PROGRAM main
  VAR
    Emergency_PB AT %IX0.0 : BOOL;
    Start_PB AT %IX0.1 : BOOL;
    Stop_PB AT %IX0.2 : BOOL;
    Fill_PositionSensor AT %IX0.4 : BOOL;
    Fill_LevelSensor AT %IX0.5 : BOOL;
    Cap_PresentSensor AT %IX0.6 : BOOL;
    NA_LabelSensor AT %IX0.7 : BOOL;
    To_M_Conv_Sensor AT %IX1.0 : BOOL;
    CaseFull_Sensor AT %IX1.1 : BOOL;
    M0 AT %IX1.2 : BOOL;
    M1 AT %IX1.3 : BOOL;
    Safety_Trip AT %IX1.4 : BOOL;
    Fill_Active AT %IX1.5 : BOOL;
    Label_PositionSensor AT %IX1.6 : BOOL;
    Reset_PB AT %IX1.7 : BOOL;
    InfeedConv_M AT %QX0.0 : BOOL;
    MainConv_M AT %QX0.1 : BOOL;
    FillValve AT %QX0.2 : BOOL;
    CapHead_M AT %QX0.3 : BOOL;
    LabelApplicator_M AT %QX0.4 : BOOL;
    RejectAcctuator_1 AT %QX0.5 : BOOL;
    RejectAcctuator_2 AT %QX0.6 : BOOL;
    TransferAcctuator AT %QX0.7 : BOOL;
    CasePacker_M AT %QX1.0 : BOOL;
    StackLight_Green AT %QX1.1 : BOOL;
    StackLight_Red AT %QX1.2 : BOOL;
    StackLight_Yellow AT %QX1.3 : BOOL;
    Alarm_Buzzer AT %QX1.4 : BOOL;
    Siren AT %QX1.5 : BOOL;
    TP0 : TP;
    TP1 : TP;
    TP2 : TP;
    TP3 : TP;
    CTU0 : CTU;
    TON0 : TON;
    TON1 : TON;
    TON2 : TON;
    RS0 : RS;
    RS1 : RS;
    RS2 : RS;
  END_VAR

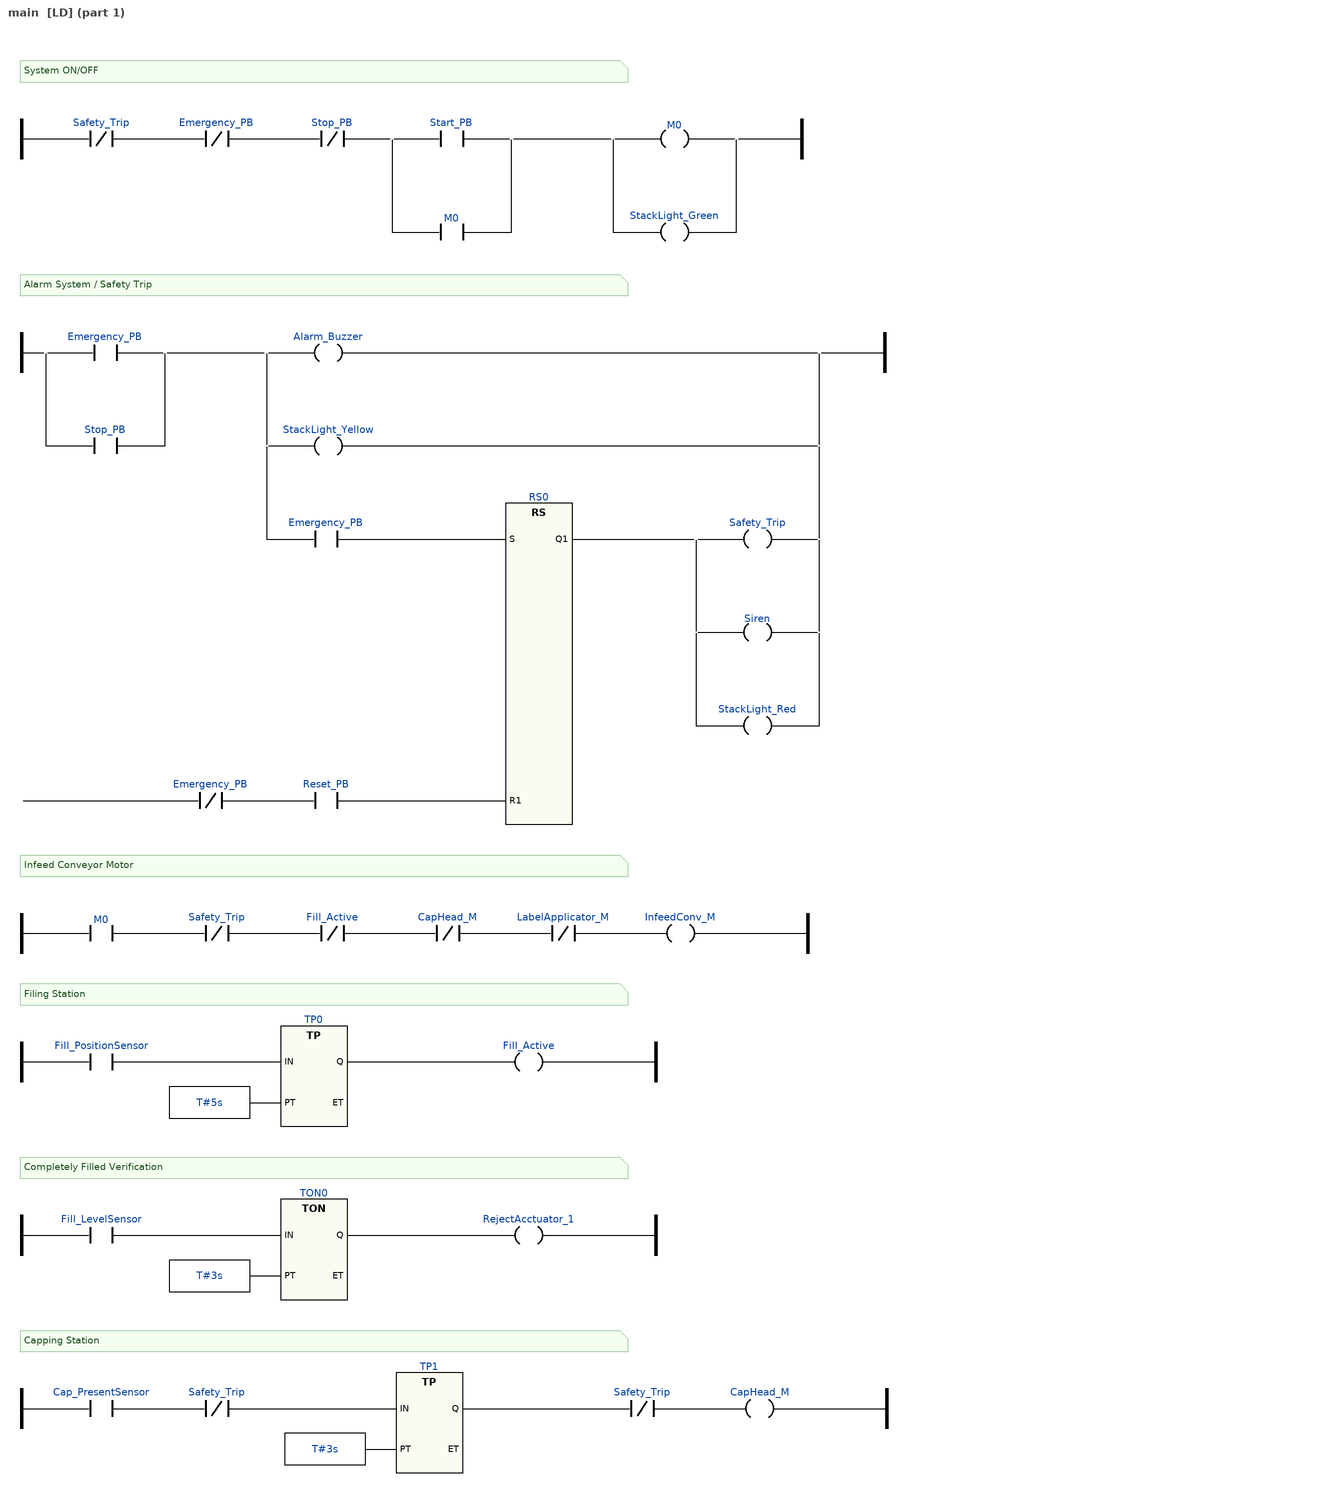
(* LD diagram, written out as Structured Text *)
(* System ON/OFF *)
M0 := NOT Safety_Trip AND NOT Emergency_PB AND NOT Stop_PB AND (Start_PB OR M0);
StackLight_Green := NOT Safety_Trip AND NOT Emergency_PB AND NOT Stop_PB AND (Start_PB OR M0);
(* Alarm System / Safety Trip *)
Alarm_Buzzer := Emergency_PB OR Stop_PB;
StackLight_Yellow := Emergency_PB OR Stop_PB;
RS0(S := (Emergency_PB OR Stop_PB) AND Emergency_PB, R1 := NOT Emergency_PB AND Reset_PB);
Safety_Trip := RS0.Q1;
Siren := RS0.Q1;
StackLight_Red := RS0.Q1;
(* Infeed Conveyor Motor *)
InfeedConv_M := M0 AND NOT Safety_Trip AND NOT Fill_Active AND NOT CapHead_M AND NOT LabelApplicator_M;
(* Filing Station *)
TP0(IN := Fill_PositionSensor, PT := T#5s);
Fill_Active := TP0.Q;
(* Completely Filled Verification *)
TON0(IN := Fill_LevelSensor, PT := T#3s);
RejectAcctuator_1 := TON0.Q;
(* Capping Station *)
TP1(IN := Cap_PresentSensor AND NOT Safety_Trip, PT := T#3s);
CapHead_M := TP1.Q AND NOT Safety_Trip;
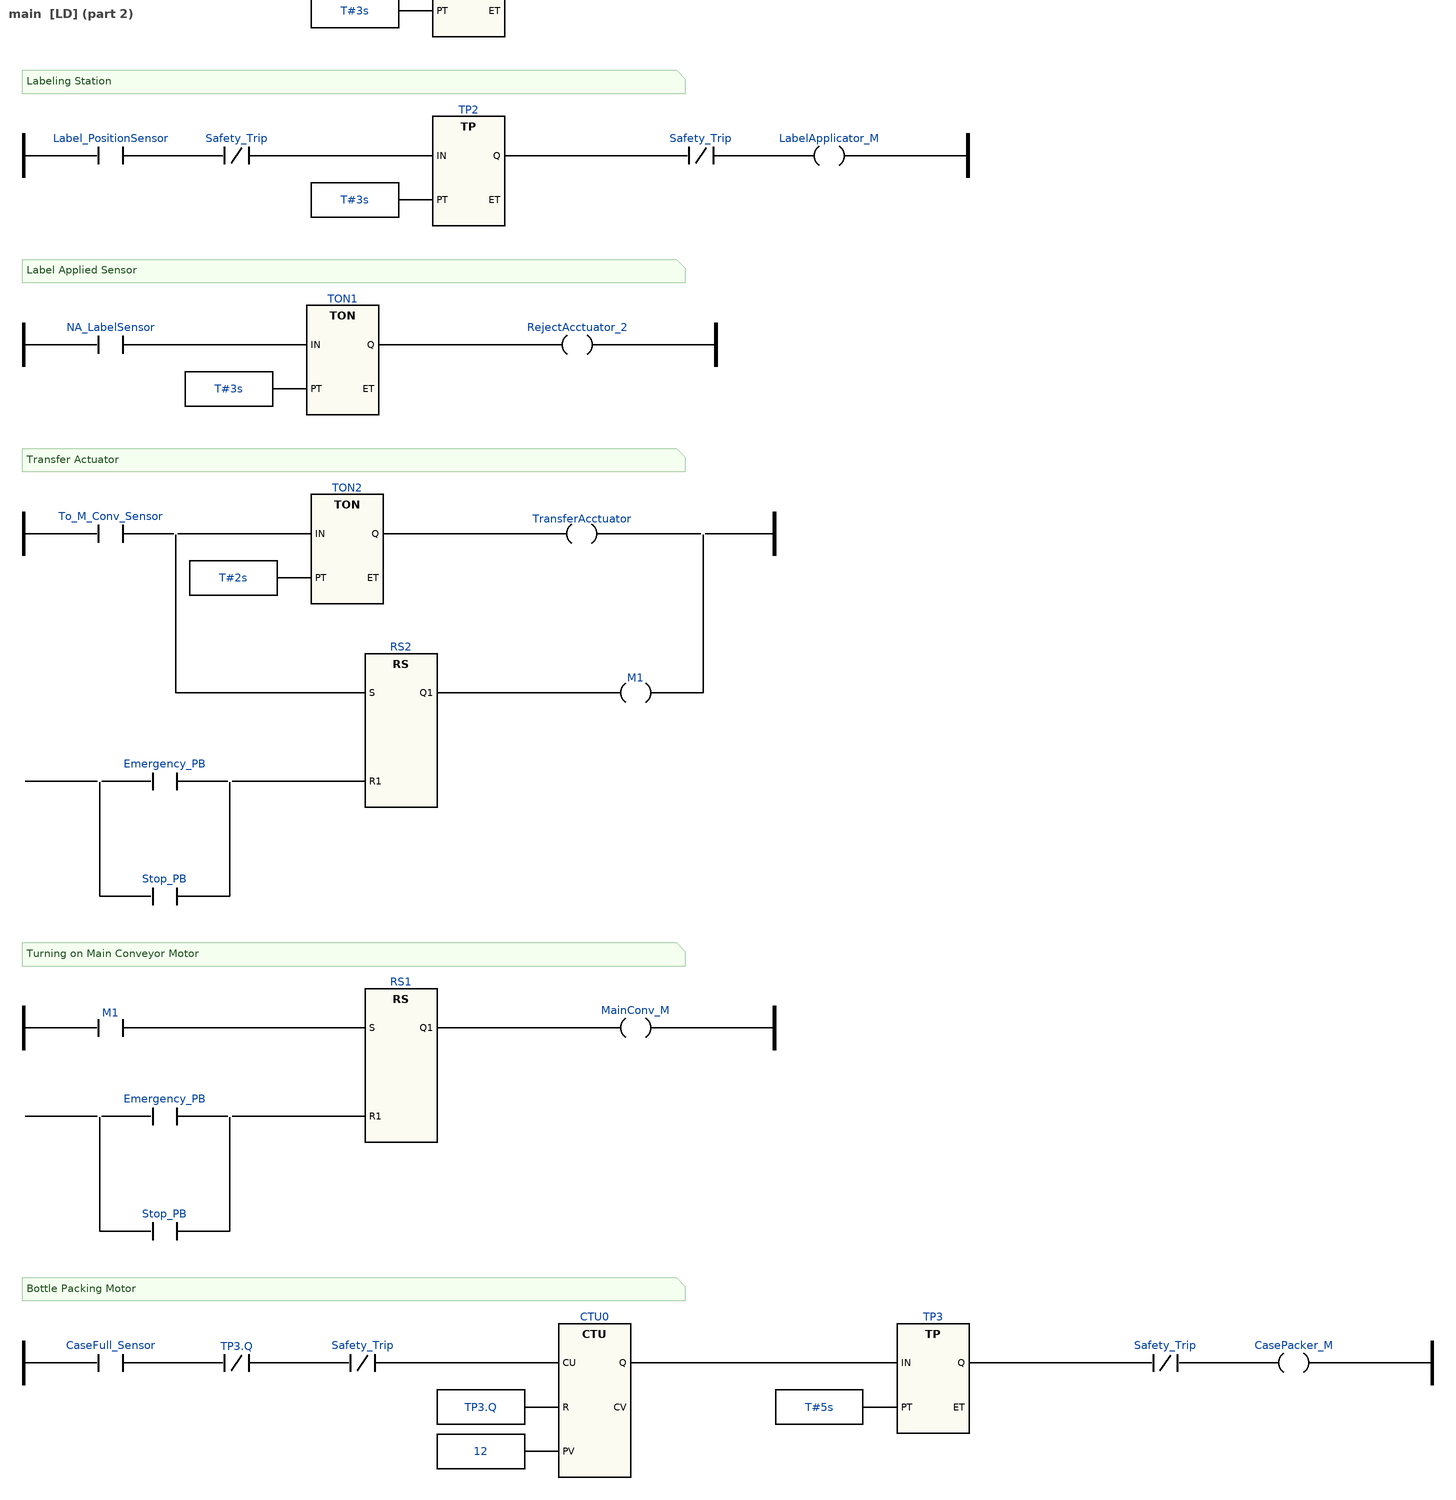
(* Labeling Station *)
TP2(IN := Label_PositionSensor AND NOT Safety_Trip, PT := T#3s);
LabelApplicator_M := TP2.Q AND NOT Safety_Trip;
(* Label Applied Sensor *)
TON1(IN := NA_LabelSensor, PT := T#3s);
RejectAcctuator_2 := TON1.Q;
(* Transfer Actuator *)
TON2(IN := To_M_Conv_Sensor, PT := T#2s);
TransferAcctuator := TON2.Q;
RS2(S := To_M_Conv_Sensor, R1 := Emergency_PB OR Stop_PB);
M1 := RS2.Q1;
(* Turning on Main Conveyor Motor *)
RS1(S := M1, R1 := Emergency_PB OR Stop_PB);
MainConv_M := RS1.Q1;
(* Bottle Packing Motor *)
CTU0(CU := CaseFull_Sensor AND NOT TP3.Q AND NOT Safety_Trip, R := TP3.Q, PV := 12);
TP3(IN := CTU0.Q, PT := T#5s);
CasePacker_M := TP3.Q AND NOT Safety_Trip;
END_PROGRAM
